// TIA Portal V20 export
TYPE "typeCmInterface"
// stored: Access Published, Namespace Unit1.Em7
   STRUCT
      brakeTest : "Unit1.Em7.typeCmInterfaceBrakeTest";
   END_STRUCT;
END_TYPE
